{attribute 'GeneratedUsingTerminal: EL2872-0000-0016'}
{attribute addProperty BoxType "EL2872-0000-0016"}
{attribute addProperty Id "EtcSlaveTerminalBaseChannel_1AT %Q*Channel_42CA91F71Channel_2AT %Q*Channel_42CA91F71Channel_3AT %Q*Channel_42CA91F71Channel_4AT %Q*Channel_42CA91F71Channel_5AT %Q*Channel_42CA91F71Channel_6AT %Q*Channel_42CA91F71Channel_7AT %Q*Channel_42CA91F71Channel_8AT %Q*Channel_42CA91F71Channel_9AT %Q*Channel_42CA91F71Channel_10AT %Q*Channel_42CA91F71Channel_11AT %Q*Channel_42CA91F71Channel_12AT %Q*Channel_42CA91F71Channel_13AT %Q*Channel_42CA91F71Channel_14AT %Q*Channel_42CA91F71Channel_15AT %Q*Channel_42CA91F71Channel_16AT %Q*Channel_42CA91F71WcStateAT %I*WcState_0B2B16F91InfoDataAT %I*InfoData_6F19DB2B2"}
{attribute addProperty CRC "3825822370"}
{attribute addProperty Size "19"}
TYPE EL2872_E4096AA2 EXTENDS EtcSlaveTerminalBase :
STRUCT
	{attribute addProperty Name "Channel_1"}
	Channel_1 : Channel_42CA91F7;
	{attribute addProperty Name "Channel_2"}
	Channel_2 : Channel_42CA91F7;
	{attribute addProperty Name "Channel_3"}
	Channel_3 : Channel_42CA91F7;
	{attribute addProperty Name "Channel_4"}
	Channel_4 : Channel_42CA91F7;
	{attribute addProperty Name "Channel_5"}
	Channel_5 : Channel_42CA91F7;
	{attribute addProperty Name "Channel_6"}
	Channel_6 : Channel_42CA91F7;
	{attribute addProperty Name "Channel_7"}
	Channel_7 : Channel_42CA91F7;
	{attribute addProperty Name "Channel_8"}
	Channel_8 : Channel_42CA91F7;
	{attribute addProperty Name "Channel_9"}
	Channel_9 : Channel_42CA91F7;
	{attribute addProperty Name "Channel_10"}
	Channel_10 : Channel_42CA91F7;
	{attribute addProperty Name "Channel_11"}
	Channel_11 : Channel_42CA91F7;
	{attribute addProperty Name "Channel_12"}
	Channel_12 : Channel_42CA91F7;
	{attribute addProperty Name "Channel_13"}
	Channel_13 : Channel_42CA91F7;
	{attribute addProperty Name "Channel_14"}
	Channel_14 : Channel_42CA91F7;
	{attribute addProperty Name "Channel_15"}
	Channel_15 : Channel_42CA91F7;
	{attribute addProperty Name "Channel_16"}
	Channel_16 : Channel_42CA91F7;
	{attribute addProperty Name "WcState"}
	WcState : WcState_0B2B16F9;
	{attribute addProperty Name "InfoData"}
	InfoData : InfoData_6F19DB2B;
END_STRUCT
END_TYPE

(* stored: Version 1.2.0.0, ProductVersion 3.1.4024.9
   DUT EL2872_E4096AA2: Id {82f1d3c6-2315-4bd9-b487-13789cc7e1a7} *)
